(* -----------------------------------------------------------------------------
| This sample has been supplied by Beckhoff As-Is and is intended only as an   |
| example implementation. Functionality is not guaranteed.                     |
----------------------------------------------------------------------------- *)

FUNCTION F_FLM_RawToLevel : REAL
VAR_INPUT
	nRaw : INT;			// valore letto dagli ingressi	
	rMaxLevel : REAL;
END_VAR
VAR_OUTPUT
    fLevel : REAL;		// [mm]	Livello
END_VAR
VAR
	
END_VAR
VAR CONSTANT
	cMAXRAW : INT := 2#0111_1111_1111_1111;	// massimo valore ingresso analogico
END_VAR

(* -----------------------------------------------------------------------------
| This sample has been supplied by Beckhoff As-Is and is intended only as an   |
| example implementation. Functionality is not guaranteed.                     |
----------------------------------------------------------------------------- *)

F_FLM_RawToLevel := (TO_REAL(nRaw) / TO_REAL(cMAXRAW)) * rMaxLevel;

END_FUNCTION

(* stored: Version 1.1.0.1, ProductVersion 3.1.4024.12
   POU F_FLM_RawToLevel: Id {ce225d20-4799-4052-92e1-3eea96198dee}, SpecialFunc None *)
